TYPE T_CRYO_PUMP_MVP030_STAT EXTENDS T_CRYO_PUMP_BASE_STAT :
STRUCT

(*
Type:
0 - old bool: 0=FALSE, NOT 0 = TRUE.
1 - UDINT
2 - REAL * 100 (with leading zeros), e.g. 001571 corresponds with 15.71
4 - STRING (6)
7 - UINT (000 to 999)

INIT commands
312 Fw version Firmware version electronic drive unit 4 R
354 HW Version Hardware version electronic drive unit 4 R
399 NominalSpd Nominal rotation speed (rpm) 1 R rpm 0 999999

STATUS commands
010 Pumpg-Statn Pump 0 = off 1 = on 0 RW 0 1 0 x
060 CtrlViaInt Operation of the interface 
	1 = remote
	2 = RS-485
	4 = PV.can
	32 = Keys on the front panel

303 Error code Error code 4 R
	Err098 Internal communication error between interface board and drive
	Err117 Vacuum pump excess temperature (> 90 °C)
	Err174 Vacuum pump blocked
	Wrn117 High temperature vacuum pump (> 75 °C)

310 DrvCurrent Drive current 2 R A 0 9999.99
311 OpHrsPump Operating hours pump 1 R h 0 65535
313 DrvVoltage Drive voltage 2 R V 0 9999.99
316 *** DrvPower Drive power 1 R W 0 999999
330 TempPump Pump temperature 1 R °C 0 999999
398 ActualSpd Actual rotation speed (rpm) 1 R rpm 0 999999

*)

// INIT commands
	sFwVersion:		STRING(8);
	sHwVersion:		STRING(8);

// STATUS commands
	sFailureCode:	STRING(8) := 'OK';
	bTargetSpeed:	BOOL;		// Target Speed Reached
	nNominalSpeed:	DINT;		// [rpm] Nominal Pump Speed
	lrMotorVolt:	LREAL;		// Pump Motor Voltage [V]

	
	bFailure:		BOOL := FALSE;	// Err of Wrn (see cmd 303)
END_STRUCT
END_TYPE

(* stored: Version 1.1.0.1, ProductVersion 3.1.4024.12
   DUT T_CRYO_PUMP_MVP030_STAT: Id {2197d692-8bad-4867-b5ff-f670c672d735} *)
